// TwinCAT 3 PLC project Inspection_Control
// ProgramVersion: 3.1.4026.20
// libraries:
//   Core, * (Beckhoff Automation LLC)
//   CoreComponents, * (Beckhoff Automation LLC)
//   CoreVision, * (Beckhoff Automation LLC)
//   Tc2_Standard, * (Beckhoff Automation GmbH)
//   Tc2_System, * (Beckhoff Automation GmbH)
//   Tc3_Vision, * (Beckhoff Automation GmbH)
// project tree:
//   GVLs/ GVL_Vision.TcGVL
//   / PlcTask.TcTTO (not stored), VisionTask.TcTTO
//   POUs/ MAIN.TcPOU, Vision.TcPOU
//   Processes/ ProcessSKU.TcPOU
//   Types/Base/ Coordinate.TcDUT, InspectionTypes.TcDUT, SystemControl.TcDUT
//   Types/Camera/ CameraRecipe.TcDUT
//   Types/Cavity/ CavityRecipe.TcDUT
//   Types/Inspections/ WaferInspection.TcDUT
//   Types/SKUs/ NestleProducts.TcDUT, SKURecipe.TcDUT
//   Types/Vision/ WaferDetectionVisionRecipe.TcDUT
//   Types/Wafer/ WaferRecipe.TcDUT
// real-time tasks:
//   TASK PlcTask: cycle T#10ms, priority 20, ADS port 350
//   TASK VisionTask: cycle T#10ms, priority 1, ADS port 351
//   TASK VnTask ImgAcq (FileSource1): cycle T#10ms, priority 5, ADS port 352

CONFIGURATION Inspection_Control
    RESOURCE PLC ON TwinCAT3
        TASK VisionTask(INTERVAL := T#10ms, PRIORITY := 1);
        PROGRAM Vision WITH VisionTask : Vision;
    END_RESOURCE
END_CONFIGURATION

// ---- Types/Base/Coordinate.TcDUT
TYPE Coordinate :
STRUCT
	X : LREAL;
	Y : LREAL;
END_STRUCT
END_TYPE

// ---- Types/Base/InspectionTypes.TcDUT
{attribute 'qualified_only'}
{attribute 'strict'}
{attribute 'to_string'}
TYPE InspectionTypes :
(
	WaferDetection := 0,
	WaferMould := 1
);
END_TYPE

// ---- Types/Base/SystemControl.TcDUT
TYPE SystemControl :
STRUCT
	StartUpRequest : BOOL;
	ShutdownRequest : BOOL;
	Reset : BOOL;
END_STRUCT
END_TYPE

// ---- Types/Camera/CameraRecipe.TcDUT
TYPE CameraRecipe :
STRUCT
	ExposureTime : UDINT;
	RulerLines : UDINT;
END_STRUCT
END_TYPE

// ---- Types/Cavity/CavityRecipe.TcDUT
TYPE CavityRecipe :
STRUCT
	LevelReference1 : Coordinate;
	LevelReference2 : Coordinate;
	MaxDifferenceBetweenLevels : LREAL;
	CavityWidth : UDINT;
	CavityLength : UDINT;
	EmptyCavityDepth : UDINT;
END_STRUCT
END_TYPE

// ---- Types/Inspections/WaferInspection.TcDUT
TYPE WaferInspection :
STRUCT
	SKU : SKURecipe;
	Cavities : CavityRecipe;
	Wafer : WaferRecipe;
	Camera : CameraRecipe;
END_STRUCT
END_TYPE

// ---- Types/SKUs/NestleProducts.TcDUT
{attribute 'qualified_only'}
{attribute 'strict'}
{attribute 'to_string'}
TYPE NestleProducts :
(
	KitKatChunky := 0,
	KitKat2Bar := 1
);
END_TYPE

// ---- Types/SKUs/SKURecipe.TcDUT
TYPE SKURecipe :
STRUCT
	MouldType : T_MaxString;
	MouldWidth : UDINT;
	MouldLength : UDINT;
	ProductType : NestleProducts;
	NumberBarsPerRow : UINT;
END_STRUCT
END_TYPE

// ---- Types/Vision/WaferDetectionVisionRecipe.TcDUT
TYPE WaferDetectionVisionRecipe :
STRUCT
	MedianFilterSize : UDINT;
END_STRUCT
END_TYPE

// ---- Types/Wafer/WaferRecipe.TcDUT
TYPE WaferRecipe :
STRUCT
	Name : T_MaxString;
	InspectionType : InspectionTypes;
	MaxWaferHeightFromBase : UDINT;
	MinWaferHeightFromBase : UDINT;
	PassingWaferCavityPercentage : UDINT;
	MaxNumberFailedBarsAllowed : UINT;
END_STRUCT
END_TYPE

// ---- GVLs/GVL_Vision.TcGVL
{attribute 'qualified_only'}
VAR_GLOBAL
	waferInspectionRecipe : WaferInspection;
	Camera : SimpleCamera;
	LabelProcess : ProcessSKU;
	ImageChannel : VisionChannel(Name := 'Beckhoff Camera', ImageSource := Camera, ImageProcess := LabelProcess);
END_VAR

// ---- POUs/Vision.TcPOU
PROGRAM Vision
VAR
END_VAR

GVL_Vision.ImageChannel.CyclicLogic();

END_PROGRAM

// ---- Processes/ProcessSKU.TcPOU
FUNCTION_BLOCK ProcessSKU EXTENDS ImageProcess
VAR
	workingImage : ITcVnImage;
	display : ITcVnDisplayableImage;
	VisionRecipe : WaferDetectionVisionRecipe;
	Result: CoreVision.VisionResult;
	ImageInfo: TcVnImageInfo;
	ValidRecipe : BOOL;
END_VAR

METHOD LoadRecipe : HRESULT
VAR_INPUT
	Recipe :  WaferDetectionVisionRecipe;
END_VAR
ValidRecipe := FALSE;

IF Recipe.MedianFilterSize = 0 THEN
	LoadRecipe := -1;
	RETURN;
END_IF

IF (Recipe.MedianFilterSize MOD 2) = 0 THEN
	 LoadRecipe := -2;
	 RETURN;
END_IF

VisionRecipe := Recipe;

ValidRecipe := TRUE;
END_METHOD

METHOD Process : HRESULT
VAR_INPUT
	Image	: REFERENCE TO CoreVision.ITcVnImage;
	hrPrev : HRESULT;
END_VAR
Image.GetImageInfo(ImageInfo);

IF NOT ValidRecipe THEN
	Trace.Error(Source := 'ProcessSKU', Message := 'Invlid Recipe for Vision');
	RETURN;
END_IF


hrPrev := F_VN_MedianFilter(Image, workingImage, VisionRecipe.MedianFilterSize, hrPrev);

Result := ProcessVisionResult(hrPrev);

hrPrev := F_VN_CopyIntoDisplayableImage(workingImage, display, hrPrev);
END_METHOD

END_FUNCTION_BLOCK

// ---- POUs/MAIN.TcPOU
PROGRAM MAIN
VAR
	ChannelControl : VisionChannelControl(Name := 'Beckhoff Camera Control',VisionChannel := GVL_Vision.ImageChannel);
	WaferDetectRecipe : WaferDetectionVisionRecipe;
	SystemCtrl : SystemControl;
	StartupState : INT;
	SystemReady : BOOL;
	ShutdownState : INT;
	OperatingState : INT;
	SKUDetected : BOOL;
	startTrig : R_TRIG;
	stopTrig : R_TRIG;
	skuTrigger : R_TRIG;
END_VAR

ChannelControl.CyclicLogic();

startTrig(CLK := SystemCtrl.StartUpRequest);
CASE StartupState OF
	0: //Unknown conditions
		IF SUCCEEDED(GVL_Vision.LabelProcess.LoadRecipe(WaferDetectRecipe)) THEN
			SystemReady := TRUE;
			StartupState := 1;
		END_IF
	1:
		IF startTrig.Q AND SystemReady THEN
			StartupState := 2;
		END_IF
	2:
		IF ChannelControl.StartVision() THEN
			StartupState := 1;
		END_IF
END_CASE

skuTrigger(CLK := SKUDetected);
CASE OperatingState OF 
	0:
		IF skuTrigger.Q THEN
			ChannelControl.TriggerImage();
			OperatingState := 1;
		END_IF
	1:
		IF NOT ChannelControl.ImageProcessingComplete THEN
			OperatingState := 2;
		END_IF
	2:
		IF ChannelControl.ImageProcessingComplete THEN
			IF ChannelControl.ImageProcessingCompletedSuccessfully THEN
				OperatingState := 0;
			ELSE
				OperatingState := 3;
			END_IF
		END_IF
		
		
END_CASE

stopTrig(CLK := SystemCtrl.ShutdownRequest);
CASE ShutdownState OF		
	0: //unkown conditions
		IF stopTrig.Q THEN
			ShutdownState := 1;
		END_IF
	1:
		IF ChannelControl.StopVision() THEN
			ShutdownState := 2;
		END_IF
END_CASE

END_PROGRAM
